(* Logix 5000 project; controller STAT 1756-L72 rev 20.12; software revision 20.04; part 30 of 34 *)
(* tags used below, declared in another part *)
   B3 : DINT[35];
   N20 : DINT[50];
   N7 : DINT[150];
   N9 : DINT[200];
   T4 : TIMER[100];
   stocklancy4 : DINT;   // alarme lvl 1 stock
   stocklancy5 : DINT;   // alarme lvl 2 stock
(* LANCY, continued *)

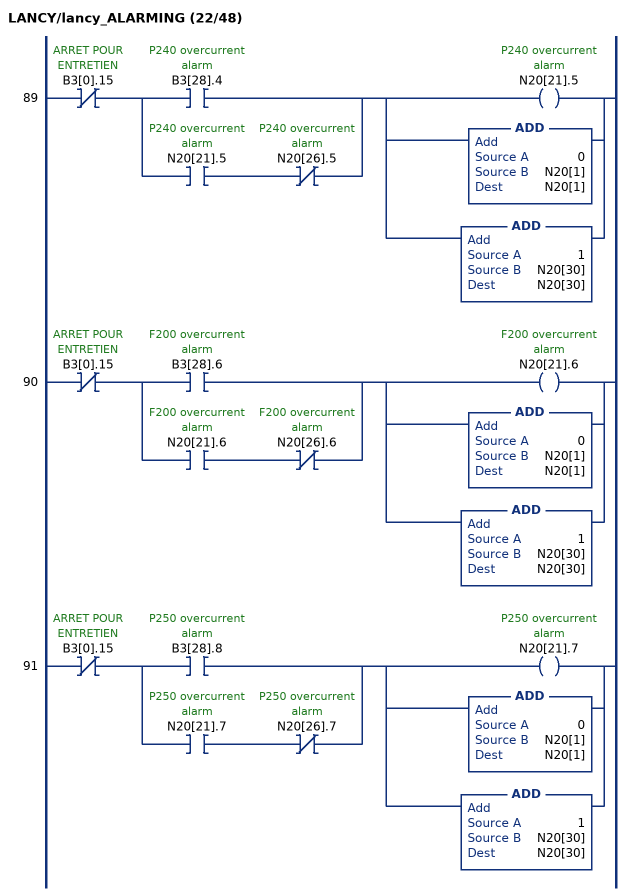
   [picture p602: LANCY/lancy_ALARMING rungs 89-91]
   89: XIO(B3[0].15)[XIC(B3[28].4) ,XIC(N20[21].5) XIO(N20[26].5) ][OTE(N20[21].5) ,ADD(0,N20[1],N20[1]) ,ADD(1,N20[30],N20[30]) ];
   90: XIO(B3[0].15)[XIC(B3[28].6) ,XIC(N20[21].6) XIO(N20[26].6) ][OTE(N20[21].6) ,ADD(0,N20[1],N20[1]) ,ADD(1,N20[30],N20[30]) ];
   91: XIO(B3[0].15)[XIC(B3[28].8) ,XIC(N20[21].7) XIO(N20[26].7) ][OTE(N20[21].7) ,ADD(0,N20[1],N20[1]) ,ADD(1,N20[30],N20[30]) ];
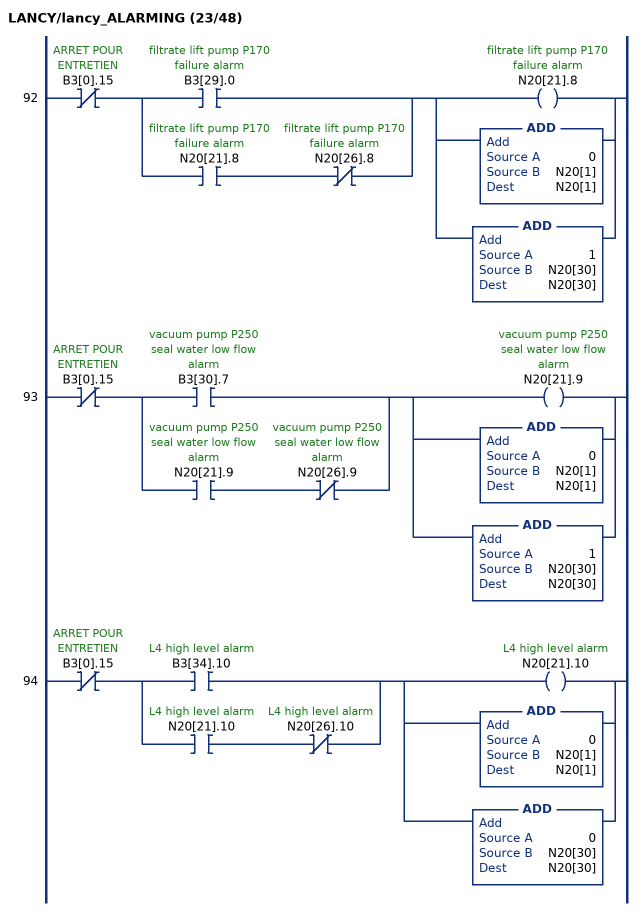
   92: XIO(B3[0].15)[XIC(B3[29].0) ,XIC(N20[21].8) XIO(N20[26].8) ][OTE(N20[21].8) ,ADD(0,N20[1],N20[1]) ,ADD(1,N20[30],N20[30]) ];
   93: XIO(B3[0].15)[XIC(B3[30].7) ,XIC(N20[21].9) XIO(N20[26].9) ][OTE(N20[21].9) ,ADD(0,N20[1],N20[1]) ,ADD(1,N20[30],N20[30]) ];
   94: XIO(B3[0].15)[XIC(B3[34].10) ,XIC(N20[21].10) XIO(N20[26].10) ][OTE(N20[21].10) ,ADD(0,N20[1],N20[1]) ,ADD(0,N20[30],N20[30]) ];
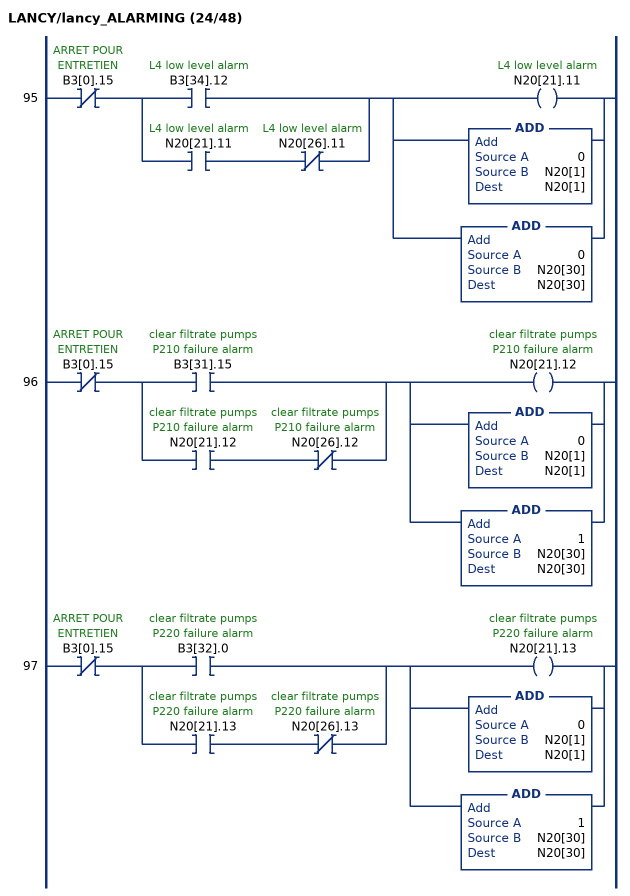
   95: XIO(B3[0].15)[XIC(B3[34].12) ,XIC(N20[21].11) XIO(N20[26].11) ][OTE(N20[21].11) ,ADD(0,N20[1],N20[1]) ,ADD(0,N20[30],N20[30]) ];
   96: XIO(B3[0].15)[XIC(B3[31].15) ,XIC(N20[21].12) XIO(N20[26].12) ][OTE(N20[21].12) ,ADD(0,N20[1],N20[1]) ,ADD(1,N20[30],N20[30]) ];
   97: XIO(B3[0].15)[XIC(B3[32].0) ,XIC(N20[21].13) XIO(N20[26].13) ][OTE(N20[21].13) ,ADD(0,N20[1],N20[1]) ,ADD(1,N20[30],N20[30]) ];
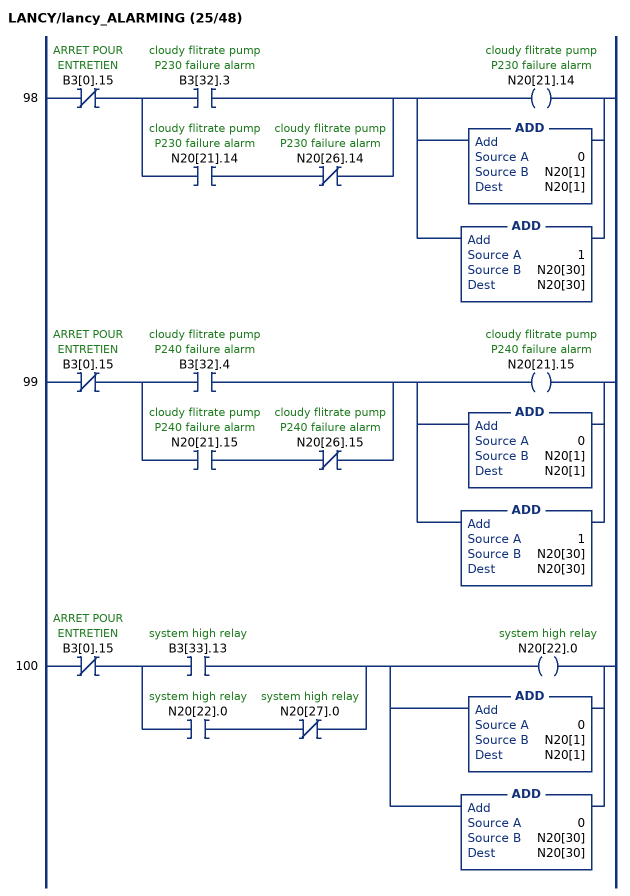
   98: XIO(B3[0].15)[XIC(B3[32].3) ,XIC(N20[21].14) XIO(N20[26].14) ][OTE(N20[21].14) ,ADD(0,N20[1],N20[1]) ,ADD(1,N20[30],N20[30]) ];
   99: XIO(B3[0].15)[XIC(B3[32].4) ,XIC(N20[21].15) XIO(N20[26].15) ][OTE(N20[21].15) ,ADD(0,N20[1],N20[1]) ,ADD(1,N20[30],N20[30]) ];
   100: XIO(B3[0].15)[XIC(B3[33].13) ,XIC(N20[22].0) XIO(N20[27].0) ][OTE(N20[22].0) ,ADD(0,N20[1],N20[1]) ,ADD(0,N20[30],N20[30]) ];
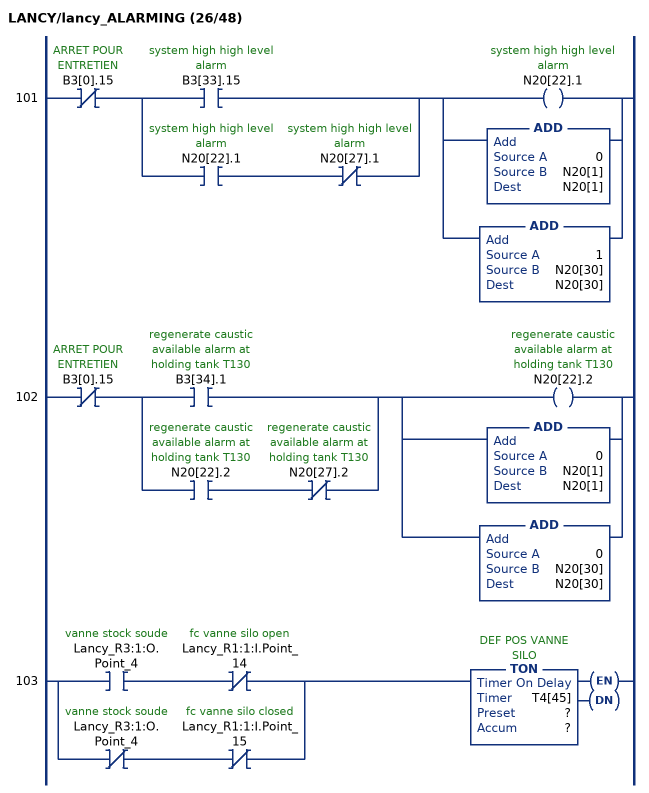
   101: XIO(B3[0].15)[XIC(B3[33].15) ,XIC(N20[22].1) XIO(N20[27].1) ][OTE(N20[22].1) ,ADD(0,N20[1],N20[1]) ,ADD(1,N20[30],N20[30]) ];
   102: XIO(B3[0].15)[XIC(B3[34].1) ,XIC(N20[22].2) XIO(N20[27].2) ][OTE(N20[22].2) ,ADD(0,N20[1],N20[1]) ,ADD(0,N20[30],N20[30]) ];
   103: [XIC(Lancy_R3:1:O.Point_4) XIO(Lancy_R1:1:I.Point_14) ,XIO(Lancy_R3:1:O.Point_4) XIO(Lancy_R1:1:I.Point_15) ]TON(T4[45],?,?);
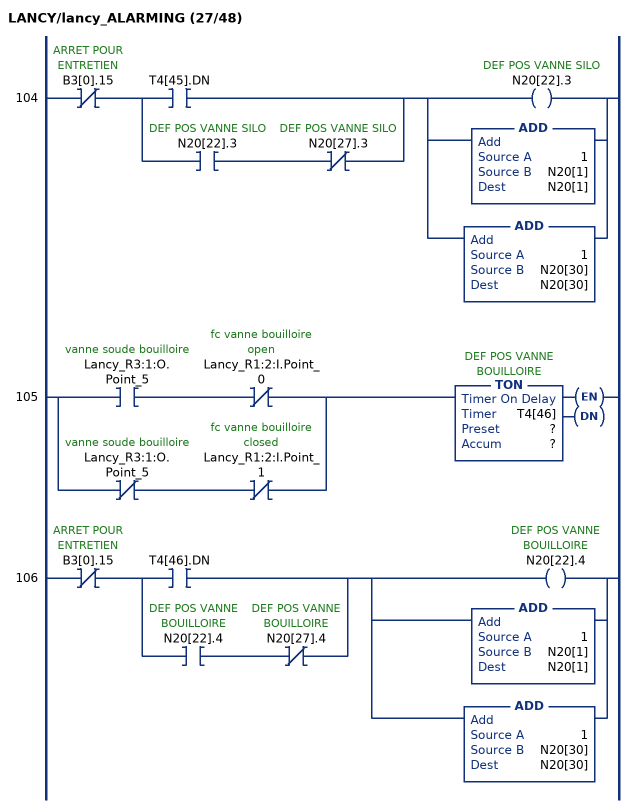
   104: XIO(B3[0].15)[XIC(T4[45].DN) ,XIC(N20[22].3) XIO(N20[27].3) ][OTE(N20[22].3) ,ADD(1,N20[1],N20[1]) ,ADD(1,N20[30],N20[30]) ];
   105: [XIC(Lancy_R3:1:O.Point_5) XIO(Lancy_R1:2:I.Point_0) ,XIO(Lancy_R3:1:O.Point_5) XIO(Lancy_R1:2:I.Point_1) ]TON(T4[46],?,?);
   106: XIO(B3[0].15)[XIC(T4[46].DN) ,XIC(N20[22].4) XIO(N20[27].4) ][OTE(N20[22].4) ,ADD(1,N20[1],N20[1]) ,ADD(1,N20[30],N20[30]) ];
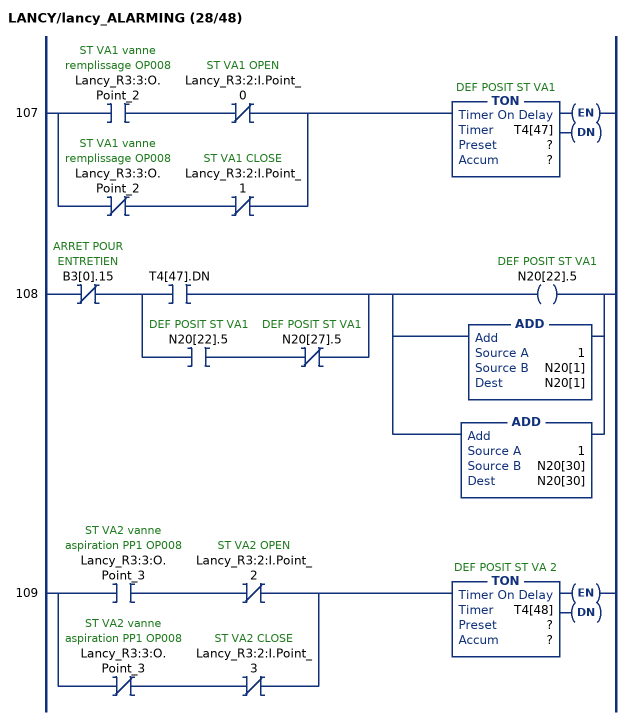
   107: [XIC(Lancy_R3:3:O.Point_2) XIO(Lancy_R3:2:I.Point_0) ,XIO(Lancy_R3:3:O.Point_2) XIO(Lancy_R3:2:I.Point_1) ]TON(T4[47],?,?);
   108: XIO(B3[0].15)[XIC(T4[47].DN) ,XIC(N20[22].5) XIO(N20[27].5) ][OTE(N20[22].5) ,ADD(1,N20[1],N20[1]) ,ADD(1,N20[30],N20[30]) ];
   109: [XIC(Lancy_R3:3:O.Point_3) XIO(Lancy_R3:2:I.Point_2) ,XIO(Lancy_R3:3:O.Point_3) XIO(Lancy_R3:2:I.Point_3) ]TON(T4[48],?,?);
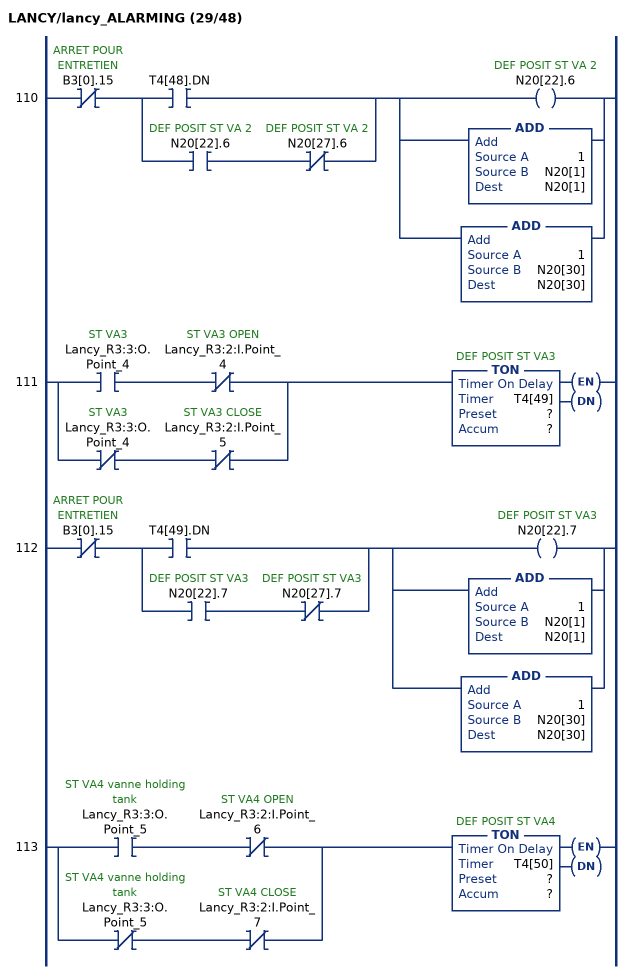
   110: XIO(B3[0].15)[XIC(T4[48].DN) ,XIC(N20[22].6) XIO(N20[27].6) ][OTE(N20[22].6) ,ADD(1,N20[1],N20[1]) ,ADD(1,N20[30],N20[30]) ];
   111: [XIC(Lancy_R3:3:O.Point_4) XIO(Lancy_R3:2:I.Point_4) ,XIO(Lancy_R3:3:O.Point_4) XIO(Lancy_R3:2:I.Point_5) ]TON(T4[49],?,?);
   112: XIO(B3[0].15)[XIC(T4[49].DN) ,XIC(N20[22].7) XIO(N20[27].7) ][OTE(N20[22].7) ,ADD(1,N20[1],N20[1]) ,ADD(1,N20[30],N20[30]) ];
   113: [XIC(Lancy_R3:3:O.Point_5) XIO(Lancy_R3:2:I.Point_6) ,XIO(Lancy_R3:3:O.Point_5) XIO(Lancy_R3:2:I.Point_7) ]TON(T4[50],?,?);
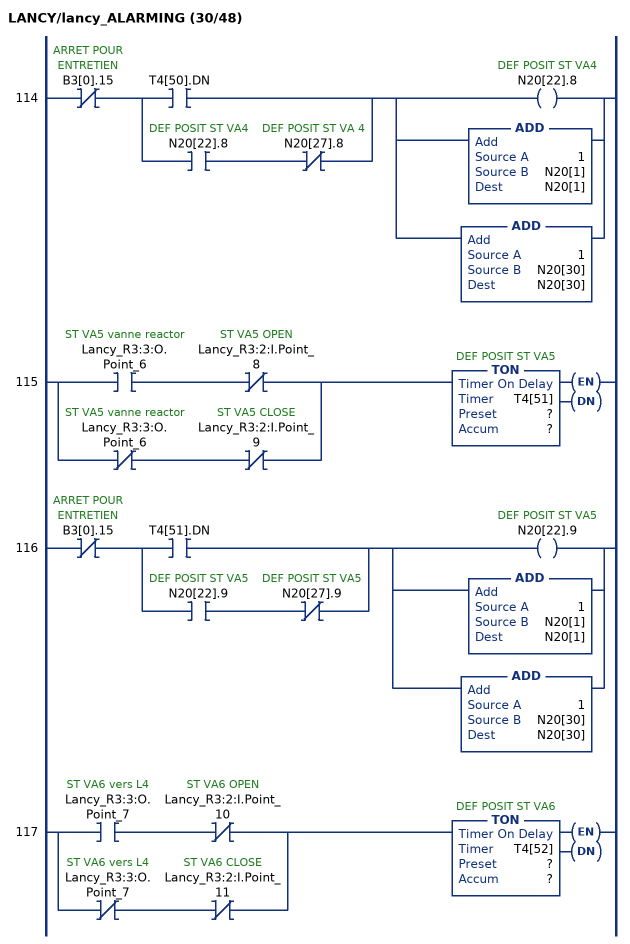
   114: XIO(B3[0].15)[XIC(T4[50].DN) ,XIC(N20[22].8) XIO(N20[27].8) ][OTE(N20[22].8) ,ADD(1,N20[1],N20[1]) ,ADD(1,N20[30],N20[30]) ];
   115: [XIC(Lancy_R3:3:O.Point_6) XIO(Lancy_R3:2:I.Point_8) ,XIO(Lancy_R3:3:O.Point_6) XIO(Lancy_R3:2:I.Point_9) ]TON(T4[51],?,?);
   116: XIO(B3[0].15)[XIC(T4[51].DN) ,XIC(N20[22].9) XIO(N20[27].9) ][OTE(N20[22].9) ,ADD(1,N20[1],N20[1]) ,ADD(1,N20[30],N20[30]) ];
   117: [XIC(Lancy_R3:3:O.Point_7) XIO(Lancy_R3:2:I.Point_10) ,XIO(Lancy_R3:3:O.Point_7) XIO(Lancy_R3:2:I.Point_11) ]TON(T4[52],?,?);
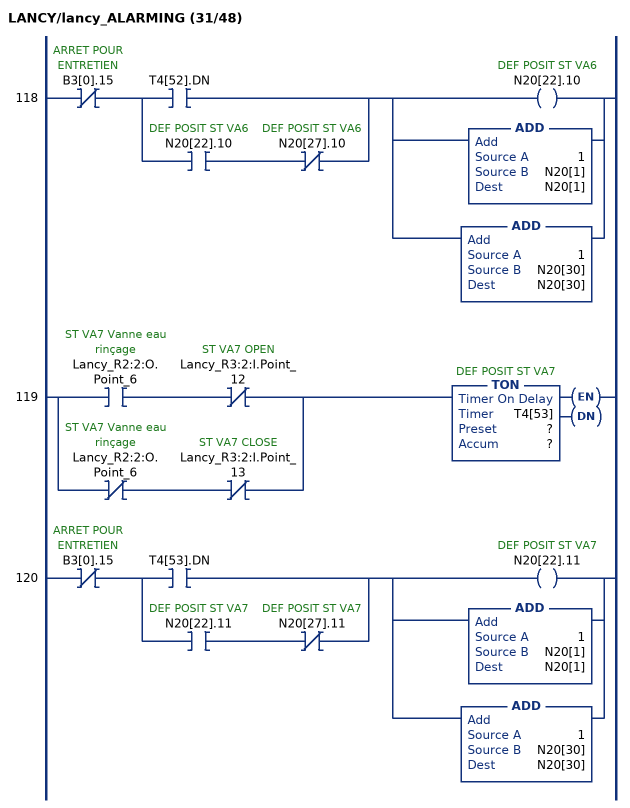
   118: XIO(B3[0].15)[XIC(T4[52].DN) ,XIC(N20[22].10) XIO(N20[27].10) ][OTE(N20[22].10) ,ADD(1,N20[1],N20[1]) ,ADD(1,N20[30],N20[30]) ];
   119: [XIC(Lancy_R2:2:O.Point_6) XIO(Lancy_R3:2:I.Point_12) ,XIO(Lancy_R2:2:O.Point_6) XIO(Lancy_R3:2:I.Point_13) ]TON(T4[53],?,?);
   120: XIO(B3[0].15)[XIC(T4[53].DN) ,XIC(N20[22].11) XIO(N20[27].11) ][OTE(N20[22].11) ,ADD(1,N20[1],N20[1]) ,ADD(1,N20[30],N20[30]) ];
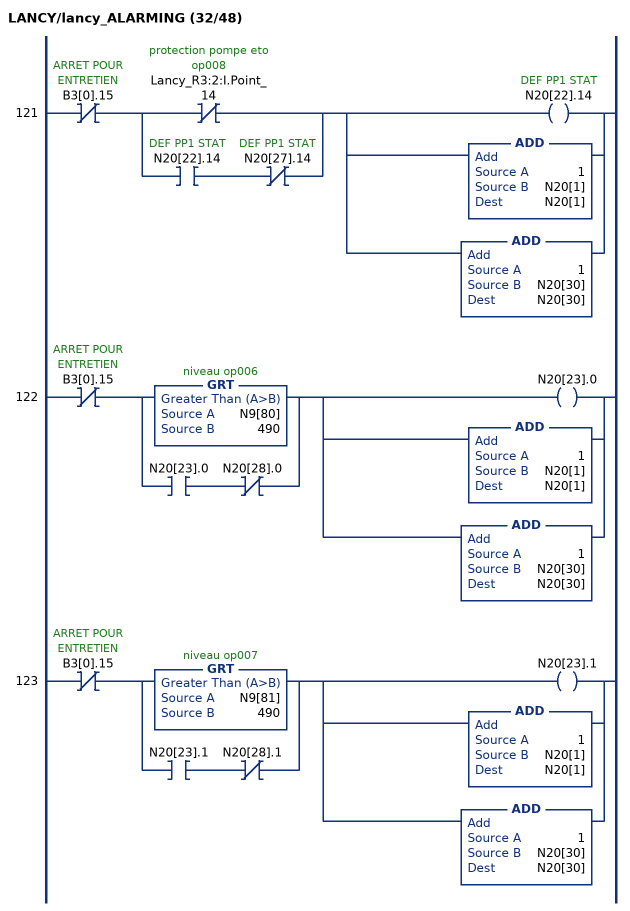
   121: XIO(B3[0].15)[XIO(Lancy_R3:2:I.Point_14) ,XIC(N20[22].14) XIO(N20[27].14) ][OTE(N20[22].14) ,ADD(1,N20[1],N20[1]) ,ADD(1,N20[30],N20[30]) ];
   122: XIO(B3[0].15)[GRT(N9[80],490) ,XIC(N20[23].0) XIO(N20[28].0) ][OTE(N20[23].0) ,ADD(1,N20[1],N20[1]) ,ADD(1,N20[30],N20[30]) ];
   123: XIO(B3[0].15)[GRT(N9[81],490) ,XIC(N20[23].1) XIO(N20[28].1) ][OTE(N20[23].1) ,ADD(1,N20[1],N20[1]) ,ADD(1,N20[30],N20[30]) ];
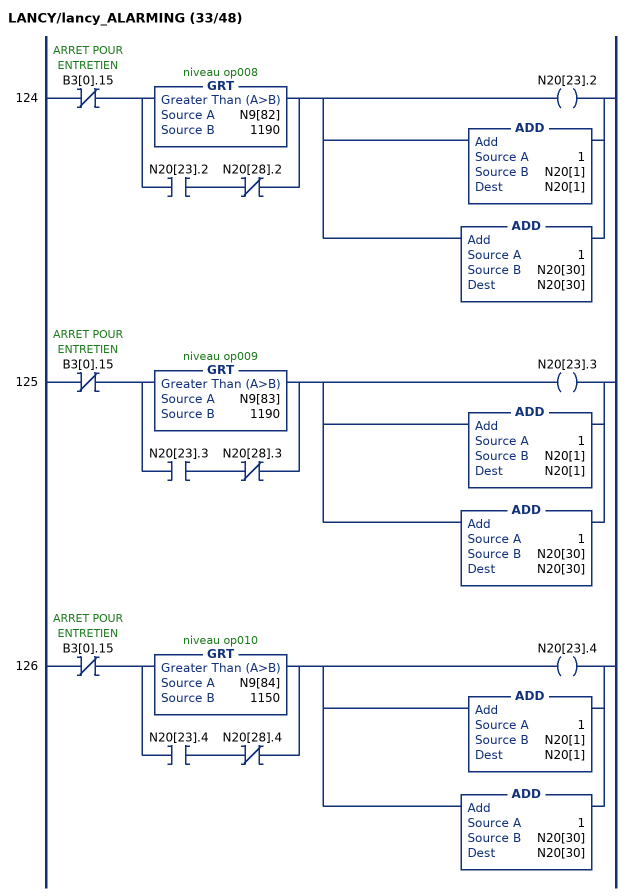
   124: XIO(B3[0].15)[GRT(N9[82],1190) ,XIC(N20[23].2) XIO(N20[28].2) ][OTE(N20[23].2) ,ADD(1,N20[1],N20[1]) ,ADD(1,N20[30],N20[30]) ];
   125: XIO(B3[0].15)[GRT(N9[83],1190) ,XIC(N20[23].3) XIO(N20[28].3) ][OTE(N20[23].3) ,ADD(1,N20[1],N20[1]) ,ADD(1,N20[30],N20[30]) ];
   126: XIO(B3[0].15)[GRT(N9[84],1150) ,XIC(N20[23].4) XIO(N20[28].4) ][OTE(N20[23].4) ,ADD(1,N20[1],N20[1]) ,ADD(1,N20[30],N20[30]) ];
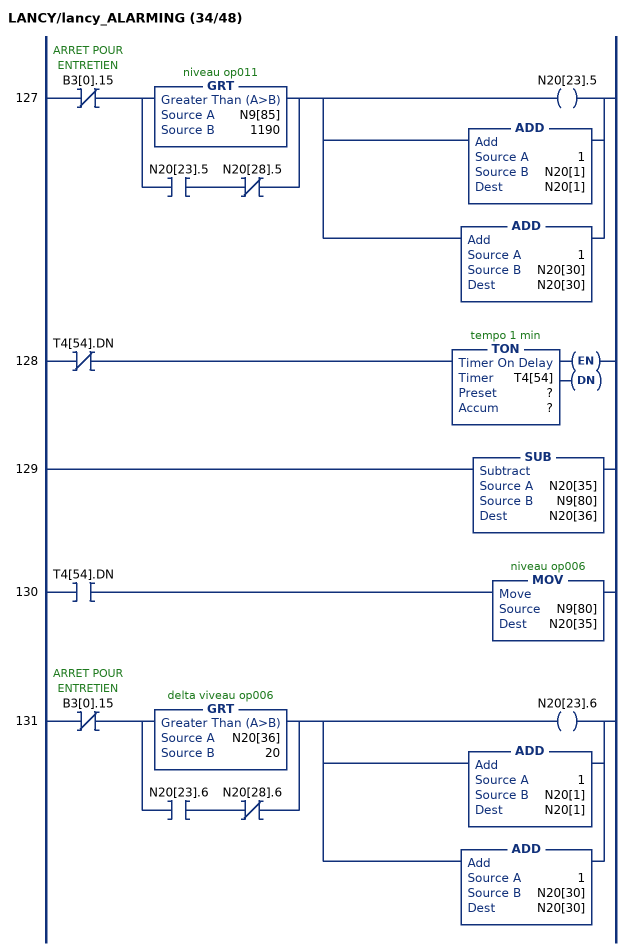
   127: XIO(B3[0].15)[GRT(N9[85],1190) ,XIC(N20[23].5) XIO(N20[28].5) ][OTE(N20[23].5) ,ADD(1,N20[1],N20[1]) ,ADD(1,N20[30],N20[30]) ];
   128: XIO(T4[54].DN)TON(T4[54],?,?);
   129: SUB(N20[35],N9[80],N20[36]);
   130: XIC(T4[54].DN)MOV(N9[80],N20[35]);
   131: XIO(B3[0].15)[GRT(N20[36],20) ,XIC(N20[23].6) XIO(N20[28].6) ][OTE(N20[23].6) ,ADD(1,N20[1],N20[1]) ,ADD(1,N20[30],N20[30]) ];
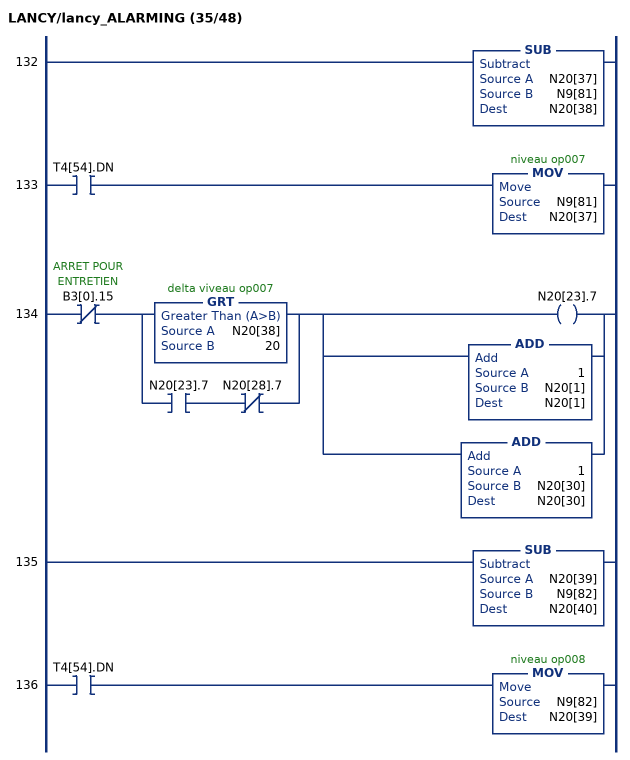
   132: SUB(N20[37],N9[81],N20[38]);
   133: XIC(T4[54].DN)MOV(N9[81],N20[37]);
   134: XIO(B3[0].15)[GRT(N20[38],20) ,XIC(N20[23].7) XIO(N20[28].7) ][OTE(N20[23].7) ,ADD(1,N20[1],N20[1]) ,ADD(1,N20[30],N20[30]) ];
   135: SUB(N20[39],N9[82],N20[40]);
   136: XIC(T4[54].DN)MOV(N9[82],N20[39]);
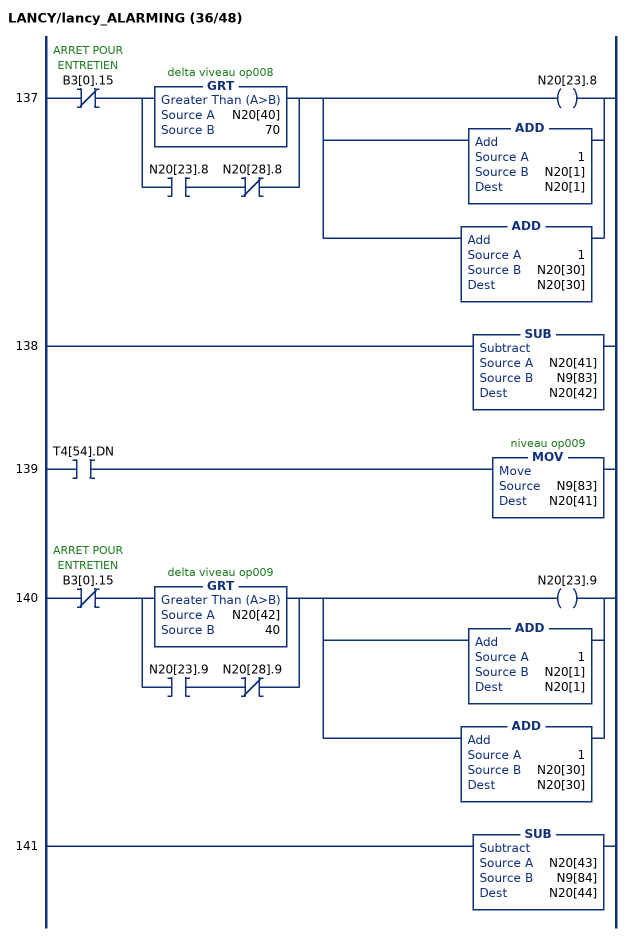
   137: XIO(B3[0].15)[GRT(N20[40],70) ,XIC(N20[23].8) XIO(N20[28].8) ][OTE(N20[23].8) ,ADD(1,N20[1],N20[1]) ,ADD(1,N20[30],N20[30]) ];
   138: SUB(N20[41],N9[83],N20[42]);
   139: XIC(T4[54].DN)MOV(N9[83],N20[41]);
   140: XIO(B3[0].15)[GRT(N20[42],40) ,XIC(N20[23].9) XIO(N20[28].9) ][OTE(N20[23].9) ,ADD(1,N20[1],N20[1]) ,ADD(1,N20[30],N20[30]) ];
   141: SUB(N20[43],N9[84],N20[44]);
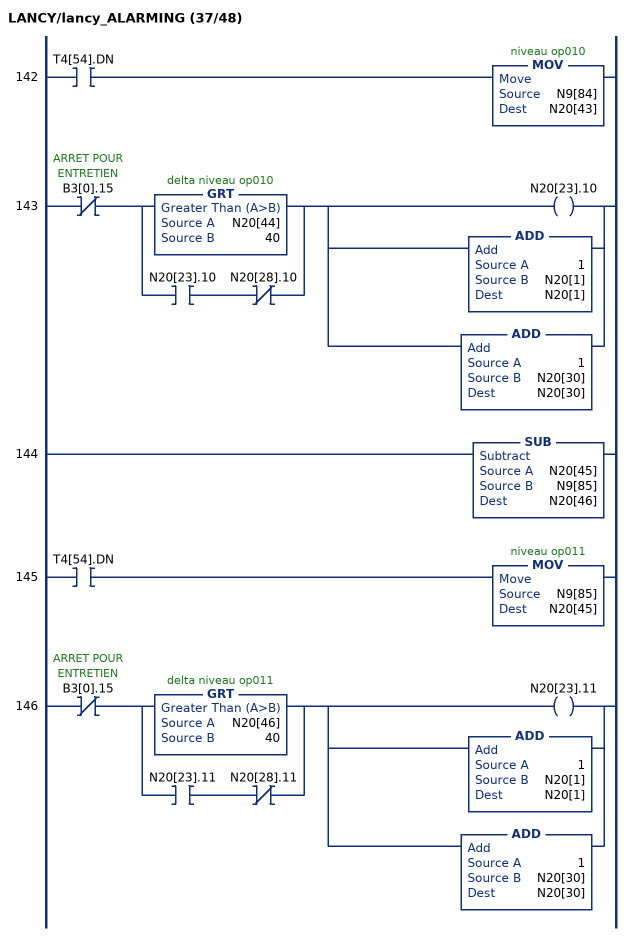
   142: XIC(T4[54].DN)MOV(N9[84],N20[43]);
   143: XIO(B3[0].15)[GRT(N20[44],40) ,XIC(N20[23].10) XIO(N20[28].10) ][OTE(N20[23].10) ,ADD(1,N20[1],N20[1]) ,ADD(1,N20[30],N20[30]) ];
   144: SUB(N20[45],N9[85],N20[46]);
   145: XIC(T4[54].DN)MOV(N9[85],N20[45]);
   146: XIO(B3[0].15)[GRT(N20[46],40) ,XIC(N20[23].11) XIO(N20[28].11) ][OTE(N20[23].11) ,ADD(1,N20[1],N20[1]) ,ADD(1,N20[30],N20[30]) ];
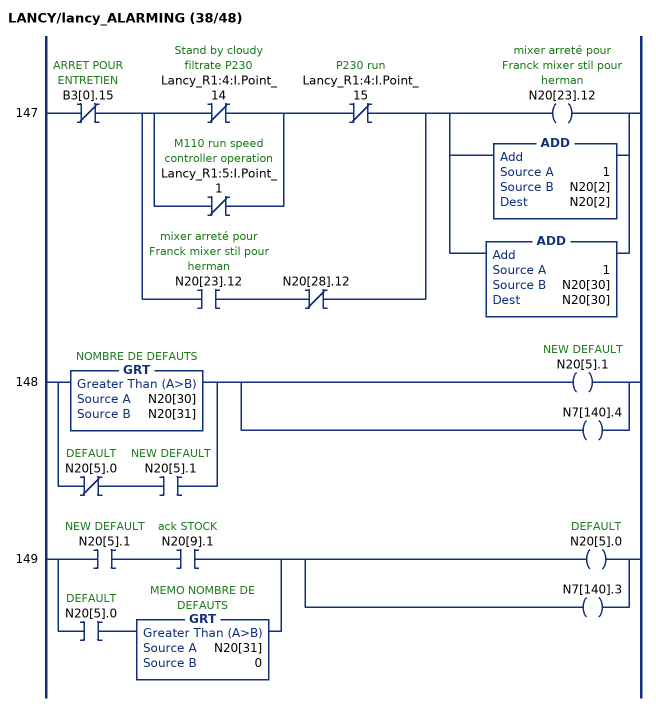
   147: XIO(B3[0].15)[[XIO(Lancy_R1:4:I.Point_14) ,XIO(Lancy_R1:5:I.Point_1) ] XIO(Lancy_R1:4:I.Point_15) ,XIC(N20[23].12) XIO(N20[28].12) ][OTE(N20[23].12) ,ADD(1,N20[2],N20[2]) ,ADD(1,N20[30],N20[30]) ];
   148: [GRT(N20[30],N20[31]) ,XIO(N20[5].0) XIC(N20[5].1) ][OTE(N20[5].1) ,OTE(N7[140].4) ];
   149: [XIC(N20[5].1) XIC(N20[9].1) ,XIC(N20[5].0) GRT(N20[31],0) ][OTE(N20[5].0) ,OTE(N7[140].3) ];
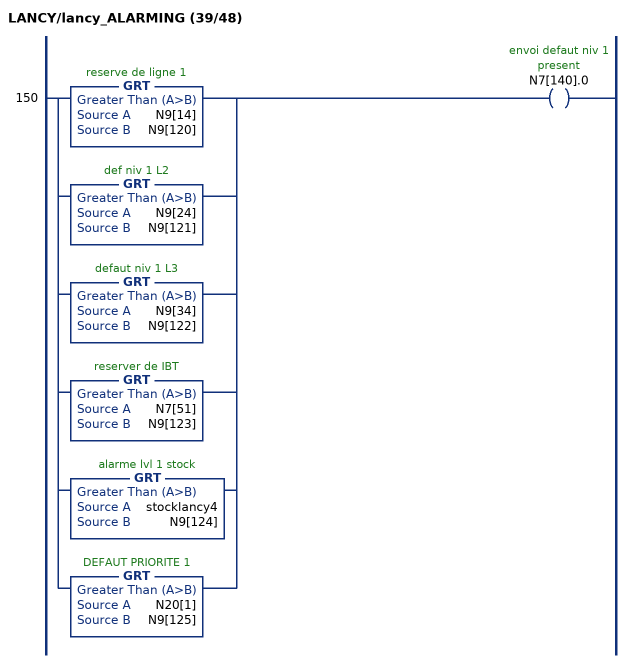
   150: [GRT(N9[14],N9[120]) ,GRT(N9[24],N9[121]) ,GRT(N9[34],N9[122]) ,GRT(N7[51],N9[123]) ,GRT(stocklancy4,N9[124]) ,GRT(N20[1],N9[125]) ]OTE(N7[140].0);
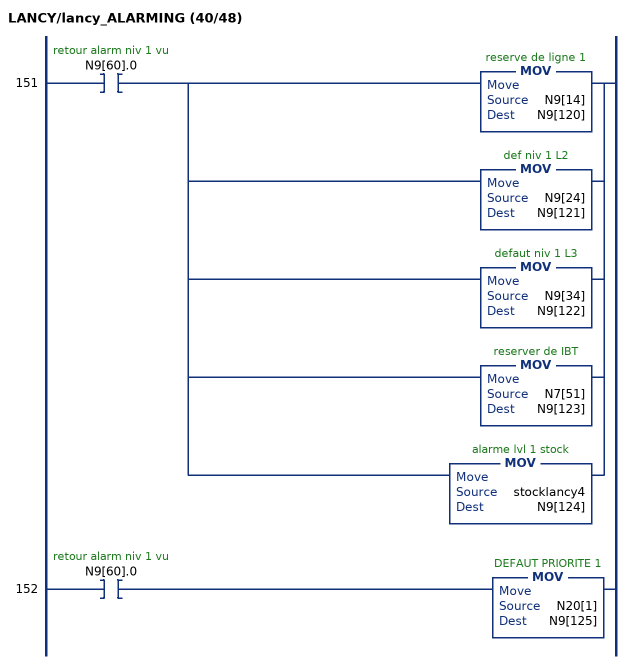
   151: XIC(N9[60].0)[MOV(N9[14],N9[120]) ,MOV(N9[24],N9[121]) ,MOV(N9[34],N9[122]) ,MOV(N7[51],N9[123]) ,MOV(stocklancy4,N9[124]) ];
   152: XIC(N9[60].0)MOV(N20[1],N9[125]);
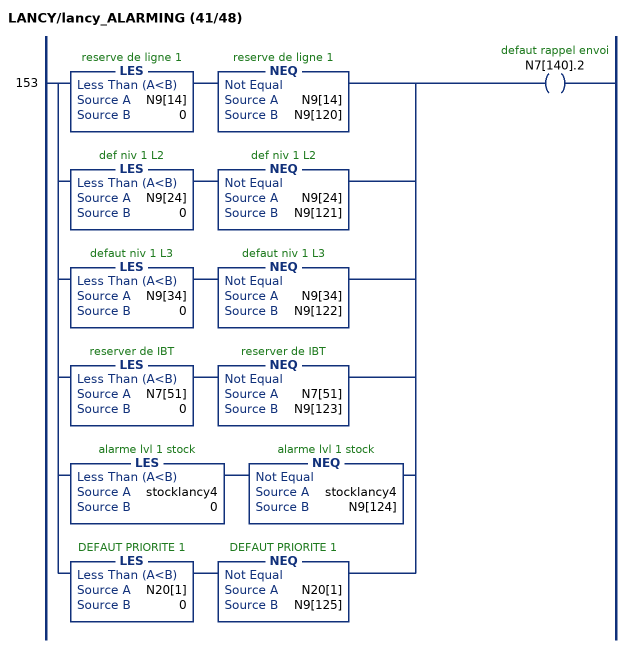
   153: [LES(N9[14],0) NEQ(N9[14],N9[120]) ,LES(N9[24],0) NEQ(N9[24],N9[121]) ,LES(N9[34],0) NEQ(N9[34],N9[122]) ,LES(N7[51],0) NEQ(N7[51],N9[123]) ,LES(stocklancy4,0) NEQ(stocklancy4,N9[124]) ,LES(N20[1],0) NEQ(N20[1],N9[125]) ]OTE(N7[140].2);
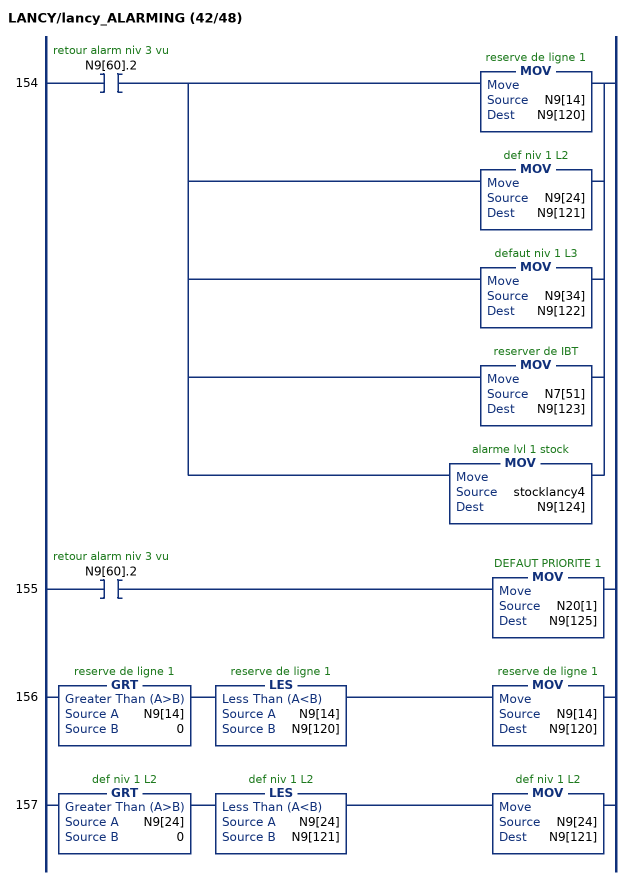
   154: XIC(N9[60].2)[MOV(N9[14],N9[120]) ,MOV(N9[24],N9[121]) ,MOV(N9[34],N9[122]) ,MOV(N7[51],N9[123]) ,MOV(stocklancy4,N9[124]) ];
   155: XIC(N9[60].2)MOV(N20[1],N9[125]);
   156: GRT(N9[14],0)LES(N9[14],N9[120])MOV(N9[14],N9[120]);
   157: GRT(N9[24],0)LES(N9[24],N9[121])MOV(N9[24],N9[121]);
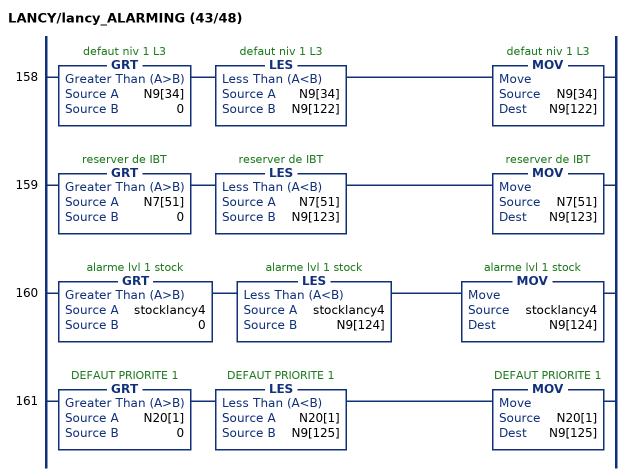
   158: GRT(N9[34],0)LES(N9[34],N9[122])MOV(N9[34],N9[122]);
   159: GRT(N7[51],0)LES(N7[51],N9[123])MOV(N7[51],N9[123]);
   160: GRT(stocklancy4,0)LES(stocklancy4,N9[124])MOV(stocklancy4,N9[124]);
   161: GRT(N20[1],0)LES(N20[1],N9[125])MOV(N20[1],N9[125]);
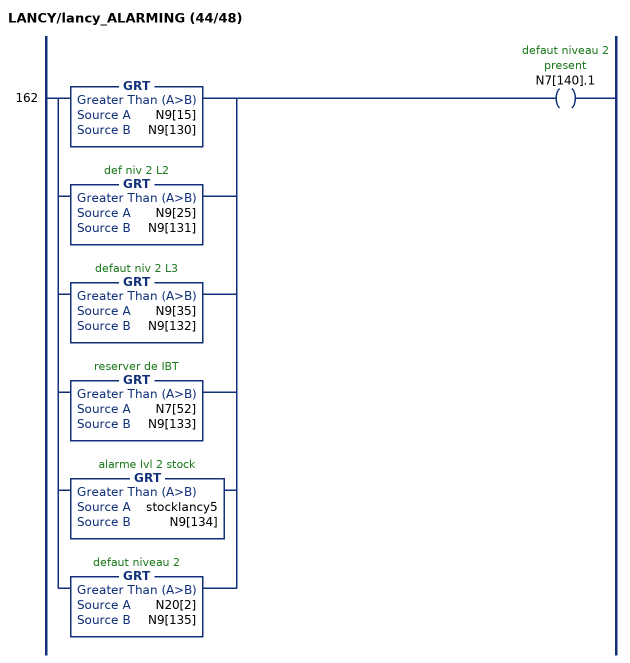
   162: [GRT(N9[15],N9[130]) ,GRT(N9[25],N9[131]) ,GRT(N9[35],N9[132]) ,GRT(N7[52],N9[133]) ,GRT(stocklancy5,N9[134]) ,GRT(N20[2],N9[135]) ]OTE(N7[140].1);
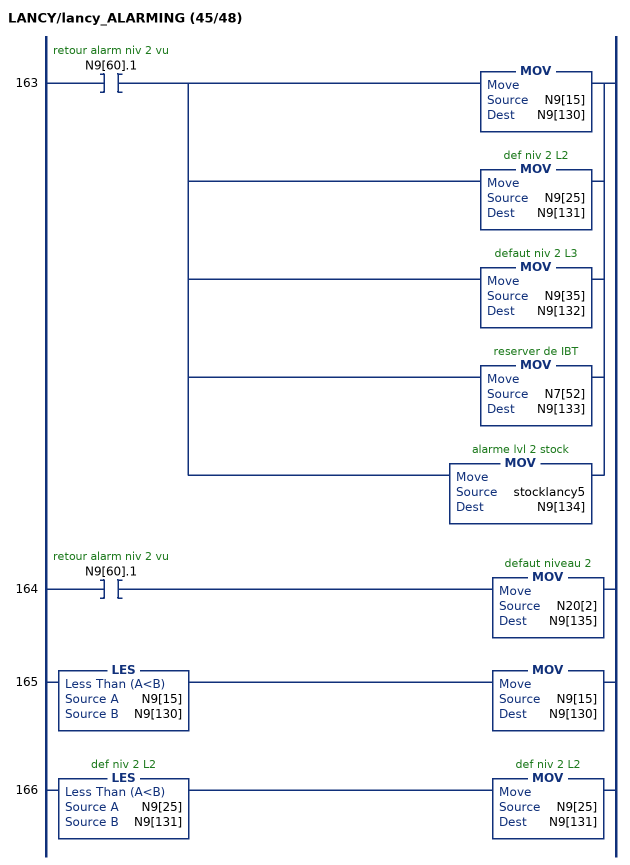
   163: XIC(N9[60].1)[MOV(N9[15],N9[130]) ,MOV(N9[25],N9[131]) ,MOV(N9[35],N9[132]) ,MOV(N7[52],N9[133]) ,MOV(stocklancy5,N9[134]) ];
   164: XIC(N9[60].1)MOV(N20[2],N9[135]);
   165: LES(N9[15],N9[130])MOV(N9[15],N9[130]);
   166: LES(N9[25],N9[131])MOV(N9[25],N9[131]);
